FUNCTION_BLOCK GO_TO_END
VAR_INPUT
END_VAR
VAR_OUTPUT
END_VAR
VAR
END_VAR

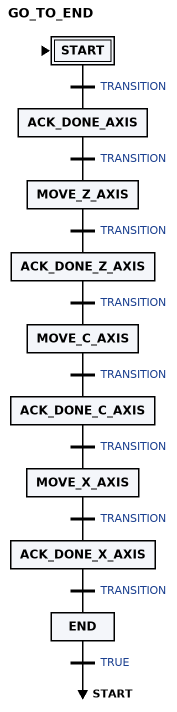
INITIAL_STEP START:
END_STEP
TRANSITION FROM START TO ACK_DONE_AXIS
    := TRANSITION;
END_TRANSITION
STEP ACK_DONE_AXIS:
END_STEP
TRANSITION FROM ACK_DONE_AXIS TO MOVE_Z_AXIS
    := TRANSITION;
END_TRANSITION
STEP MOVE_Z_AXIS:
END_STEP
TRANSITION FROM MOVE_Z_AXIS TO ACK_DONE_Z_AXIS
    := TRANSITION;
END_TRANSITION
STEP ACK_DONE_Z_AXIS:
END_STEP
TRANSITION FROM ACK_DONE_Z_AXIS TO MOVE_C_AXIS
    := TRANSITION;
END_TRANSITION
STEP MOVE_C_AXIS:
END_STEP
TRANSITION FROM MOVE_C_AXIS TO ACK_DONE_C_AXIS
    := TRANSITION;
END_TRANSITION
STEP ACK_DONE_C_AXIS:
END_STEP
TRANSITION FROM ACK_DONE_C_AXIS TO MOVE_X_AXIS
    := TRANSITION;
END_TRANSITION
STEP MOVE_X_AXIS:
END_STEP
TRANSITION FROM MOVE_X_AXIS TO ACK_DONE_X_AXIS
    := TRANSITION;
END_TRANSITION
STEP ACK_DONE_X_AXIS:
END_STEP
TRANSITION FROM ACK_DONE_X_AXIS TO END
    := TRANSITION;
END_TRANSITION
STEP END:
END_STEP
TRANSITION FROM END TO START
    := TRUE;
END_TRANSITION

TRANSITION TRANSITION:

END_TRANSITION

END_FUNCTION_BLOCK

(* stored: Version 1.1.0.1, ProductVersion 3.1.4022.18
   POU GO_TO_END: Id {038d5059-ea58-4535-9507-7965441c5abd}, SpecialFunc None
   Transition TRANSITION: Id {175e5c28-bbd1-44f7-95d5-d8036e845ea7} *)
